// TIA Portal project "P01_From_A_to_B_FIO_TMP" (V16)
// Vorlageprojekt für das Buch mit Zielsystem S7-1200

(* hardware
DEVICE "S7-1200-Station_1"  S7-1200 Station
   slot 0: "Baugruppenträger_0"  Rack  V1.0
   slot 1: "PLC_1"  CPU 1211C DC/DC/DC  6ES7 211-1AE40-0XB0  V4.1
*)

// ===== PLC "PLC_1"  CPU 1211C DC/DC/DC =====

VAR_GLOBAL   // PLC tag table "Input_Tags"
   "Photo_Sensor" AT %I0.0 : Bool;   // TRUE = Beam Clear (No Box); FALSE = Beam Blocked (Box detected)
   "Factory_Running" AT %I0.1 : Bool;   // TRUE = Simulation Running; FALSE = Simulation Stopped
   "Start_Button" AT %I0.2 : Bool;   // TRUE = Pressed; FALSE = Released
   "Stop_Button" AT %I0.3 : Bool;   // TRUE = Released; FALSE = Pressed
   "Run_Command" AT %M0.0 : Bool;   // TRUE = Conveyor Enabled; FALSE = Conveyor Disabled
END_VAR

VAR_GLOBAL   // PLC tag table "Output_Tags"
   "Conveyor_Motor" AT %Q0.0 : Bool;   // TRUE = Conveyor Running; FALSE = Conveyor Stopped
END_VAR

VAR_GLOBAL   // PLC tag table "Internal_tags"
   "Fault" AT %M0.1 : Bool;   // TRUE = Fault Active; FALSE = No Fault
   "Cycle_Start" AT %M0.2 : Bool;   // TRUE = Automatic Cycle Active; FALSE = Automatic Cycle Inactive
END_VAR

FUNCTION "FC10_Main" : Void   // FC1, LAD
{ S7_Optimized_Access := 'TRUE' }
VERSION : 0.1
BEGIN

REGION Network 1
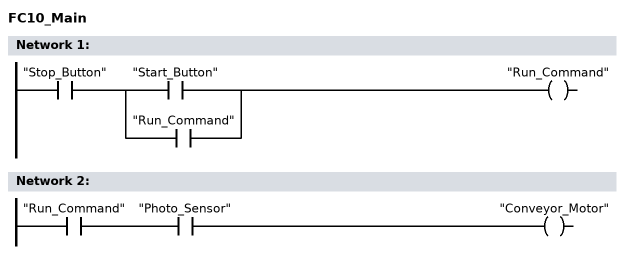
   RUNG wire#powerrail
      Contact( "Stop_Button" )
      wire#w1
      Contact( "Start_Button" )
      wire#w2
      Coil( "Run_Command" )
   END_RUNG
   RUNG wire#w1
      Contact( "Run_Command" )
   END_RUNG wire#w2
   // the same network as SCL:
   "Run_Command" := "Stop_Button" AND ("Start_Button" OR "Run_Command");
END_REGION

REGION Network 2
   RUNG wire#powerrail
      Contact( "Run_Command" )
      Contact( "Photo_Sensor" )
      Coil( "Conveyor_Motor" )
   END_RUNG
   // the same network as SCL:
   "Conveyor_Motor" := "Run_Command" AND "Photo_Sensor";
END_REGION
END_FUNCTION

FUNCTION "MHJ-PLC-Lab-Function-S71200" : Void   // FC9000, SCL
{ S7_Optimized_Access := 'TRUE' }
VERSION : 0.1
   VAR_TEMP
      rdTimeReturn : Int;
      outputTime : DTL;
      SyncVal : Byte;
      forVal : Int;
      forVal_2 : Int;
      Value : Byte;
   END_VAR
   VAR CONSTANT
      CompVal : Byte := 16#34;
      Value_01 : Byte := 16#11;
      Value_01_DW : DWord := 16#A165_D992;
      Value_02_DW : DWord := 16#58BE_4401;
   END_VAR
BEGIN

   #Value:=PEEK(area := 16#82,
        dbNumber := 0,
        byteOffset := 511);
   #Value := #Value + 1;

   POKE(area := 16#82,
        dbNumber := 0,
        byteOffset := 511,
        value := #Value);

   POKE(area:=16#81,
        dbNumber:=0,
        byteOffset:=1016,
        value:=#Value_01_DW);
   POKE(area := 16#81,
        dbNumber := 0,
        byteOffset := 1020,
        value := #Value_02_DW);

   POKE(area := 16#81,
        dbNumber := 0,
        byteOffset := 511,
        value := B#16#00);

   FOR #forVal := 0 TO 120 DO
       FOR #forVal_2:=0 TO 10 DO
           #rdTimeReturn:=RD_SYS_T(#outputTime);
           #rdTimeReturn := WR_SYS_T(#outputTime);
           #rdTimeReturn := RD_SYS_T(#outputTime);
           #rdTimeReturn := WR_SYS_T(#outputTime);
       END_FOR;
       #SyncVal:= PEEK(area := 16#81,
                      dbNumber := 0,
                      byteOffset := 511);
       IF #SyncVal = #CompVal THEN
          GOTO M_1;
       END_IF;
   END_FOR;
   RETURN;

   M_1:
   POKE(area := 16#81,
        dbNumber := 0,
        byteOffset := 511,
        value := B#16#0);
END_FUNCTION

ORGANIZATION_BLOCK "Main"   // OB1, LAD, ProgramCycle
TITLE = "Main Program Sweep (Cycle)"
{ S7_Optimized_Access := 'TRUE' }
VERSION : 0.1
   VAR_INPUT
      Initial_Call : Bool;   // Initial call of this OB
      Remanence : Bool;   // =True, if remanent data are available
   END_VAR
BEGIN

REGION Network 1: Konnektierungsbaustein für PLC-Lab
   // Im Netzwerk 1 wird der Konnektierungsbaustein für PLC-Lab aufgerufen.
   // Dieser Aufruf darf nicht entfernt werden!
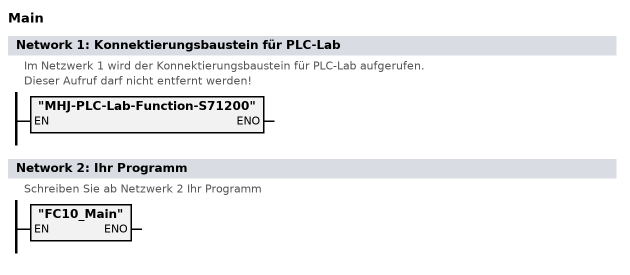
   RUNG wire#powerrail
      "MHJ-PLC-Lab-Function-S71200"()
   END_RUNG
   // the same network as SCL:
   "MHJ-PLC-Lab-Function-S71200"();
END_REGION

REGION Network 2: Ihr Programm
   // Schreiben Sie ab Netzwerk 2 Ihr Programm
   RUNG wire#powerrail
      "FC10_Main"()
   END_RUNG
   // the same network as SCL:
   "FC10_Main"();
END_REGION
END_ORGANIZATION_BLOCK